// TwinCAT 3 PLC project HutchMPS
// ProgramVersion: 3.1.4020.4
// libraries:
//   Tc2_Standard, * (Beckhoff Automation GmbH)
//   Tc2_System, * (Beckhoff Automation GmbH)
//   Tc3_Module, * (Beckhoff Automation GmbH)
// project tree:
//   GVLs/ GetBeamDemand.TcGVL
//   / PlcTask.TcTTO
//   POUs/ MAIN.TcPOU
// (motion and I/O tree: see PLC project motioncontroller)
// real-time tasks:
//   TASK PlcTask: cycle T#10ms, priority 20, ADS port 350
// variable links:

CONFIGURATION HutchMPS
    RESOURCE PLC ON TwinCAT3
        TASK PlcTask(INTERVAL := T#10ms, PRIORITY := 20);
        PROGRAM MAIN WITH PlcTask : MAIN;
    END_RESOURCE
END_CONFIGURATION

// ---- GVLs/GetBeamDemand.TcGVL
{attribute 'qualified_only'}
VAR_GLOBAL
	// What beam rate is required from a device? (Probably units of frequency) 
	beamRate	AT %I*	: LREAL;
	// Demand specifies if this demand is an emergency (True). Non-Demand is for non-emergencies/Preemtive protection (synonomous). Sent to Hutch PLC.
	// demand : BOOL;
END_VAR

// ---- POUs/MAIN.TcPOU

      PROGRAM MAIN
VAR
END_VAR

END_PROGRAM
